SYSTEM System (* System Configuration *)
  (* Standard: 61499-1 *)
  (* Version 0.0, 12/17/2022, Dmitrii, Flexbridge AB *)
  {SET_ATTRIBUTE(System.Device.FolderPath, CourierIB,CheckpointIB1,M251)}
  APPLICATION APP1
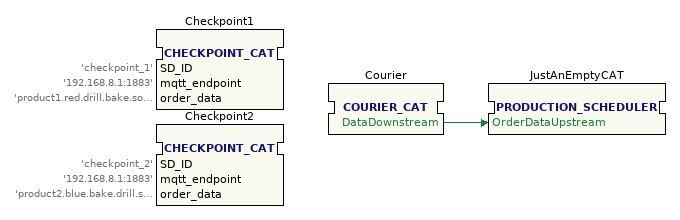
    (* Dynamic discovery here *)
    (* In case it asks for a password somwhere, thy this: Login: admin Password: UAOadmin- *)
    (* TODO place your control application here *)
    FBS
      Checkpoint1 : CHECKPOINT_CAT(SD_ID := 'checkpoint_1', mqtt_endpoint := '192.168.8.1:1883', order_data := 'product1.red.drill.bake.sort');
      Checkpoint2 : CHECKPOINT_CAT(SD_ID := 'checkpoint_2', mqtt_endpoint := '192.168.8.1:1883', order_data := 'product2.blue.bake.drill.sort');
      Courier : COURIER_CAT;
      JustAnEmptyCAT : PRODUCTION_SCHEDULER;
    END_FBS
    ADAPTER_CONNECTIONS
      Courier.DataDownstream TO JustAnEmptyCAT.OrderDataUpstream;
    END_CONNECTIONS
  END_APPLICATION
  DEVICE CourierIB : ECORT
    RESOURCE RES0 : EMB_RES_ECO
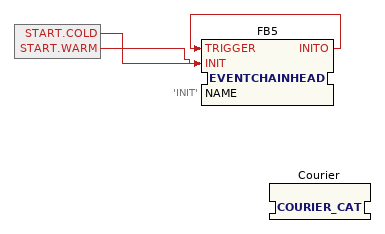
      FBS
        Courier : COURIER_CAT;
        FB5 : EVENTCHAINHEAD(NAME := 'INIT');
      END_FBS
      EVENT_CONNECTIONS
        FB5.INITO TO FB5.TRIGGER;
        START.COLD TO FB5.INIT;
        START.WARM TO FB5.INIT;
      END_CONNECTIONS
    END_RESOURCE
  END_DEVICE
  DEVICE CheckpointIB1 : ECORT
    RESOURCE RES0 : EMB_RES_ECO
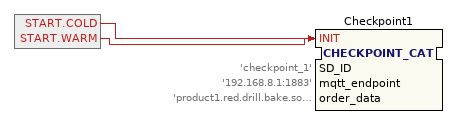
      FBS
        Checkpoint1 : CHECKPOINT_CAT(SD_ID := 'checkpoint_1', mqtt_endpoint := '192.168.8.1:1883', order_data := 'product1.red.drill.bake.sort');
      END_FBS
      EVENT_CONNECTIONS
        START.COLD TO Checkpoint1.INIT;
        START.WARM TO Checkpoint1.INIT;
      END_CONNECTIONS
    END_RESOURCE
  END_DEVICE
  DEVICE M251 : M251_dPAC
    RESOURCE RES0 : EMB_RES_ECO
      FBS
        M251_HSCAction : hscAction;
        FB1 : SYMLINKMULTIVARSRC_1559B0FF8170C9BA0(QI := TRUE, NAME1 := '$${PATH}FEn', VALUE1 := TRUE); {SET_ATTRIBUTE(Configuration.GenericFBType.InterfaceParams, Runtime.System#I:=1;VALUE${I$}:BOOL)}
        FB2 : DPAC_FULLINIT;
        FB3 : EVENTCHAINHEAD(NAME := 'INIT');
      END_FBS
      EVENT_CONNECTIONS
        M251_HSCAction.INITO TO FB1.INIT;
        START.COLD TO FB2.INIT;
        START.WARM TO FB2.INIT;
        START.ONLINECHANGE TO FB2.INIT;
        FB2.INITO TO M251_HSCAction.INIT;
        FB1.INITO TO FB3.INIT;
        FB3.INITO TO FB3.TRIGGER;
      END_CONNECTIONS
    END_RESOURCE
  END_DEVICE
  MAPPINGS
    APP1.Courier ON CourierIB.RES0;
    APP1.Checkpoint1 ON CheckpointIB1.RES0;
  END_MAPPINGS
END_SYSTEM
